// TIA Portal V20 export
VAR_GLOBAL   // PLC tag table "Spare"
   "BA010AZCRBK01.06" AT %I1000.6 : Bool;   // SPARE
   "BA010AZCRBK01.07" AT %I1000.7 : Bool;   // SPARE
   "BA010AZCRBK01.16" AT %I1001.6 : Bool;   // SPARE
   "BA010AZCRBK01.17" AT %I1001.7 : Bool;   // SPARE
   "BA010AZCRPM01.01" AT %Q2000.1 : Bool;   // SPARE
   "BA010AZCRPM01.03" AT %Q2000.3 : Bool;   // SPARE
   "BA010AZCRPM01.14" AT %Q2001.4 : Bool;   // SPARE
   "BA010AZCRPM01.15" AT %Q2001.5 : Bool;   // SPARE
   "BA010AZCRPM01.16" AT %Q2001.6 : Bool;   // SPARE
   "BA010AZCRPM01.17" AT %Q2001.7 : Bool;   // SPARE
   "BA010AZCRBK02.08" AT %I1005.0 : Bool;   // SPARE
   "BA010AZCRBK02.09" AT %I1005.1 : Bool;   // SPARE
   "BA010AZCRBK02.10" AT %I1005.2 : Bool;   // SPARE
   "BA010AZCRBK02.11" AT %I1005.3 : Bool;   // SPARE
   "BA010AZCRBK02.12" AT %I1005.4 : Bool;   // SPARE
   "BA010AZCRBK02.13" AT %I1005.5 : Bool;   // SPARE
   "BA010AZCRBK02.14" AT %I1005.6 : Bool;   // SPARE
   "BA010AZCRBK02.15" AT %I1005.7 : Bool;   // SPARE
   "BA010AZCRPM02.16" AT %Q2005.6 : Bool;   // SPARE
   "BA010AZCRPM02.17" AT %Q2005.7 : Bool;   // SPARE
   "BA010AZCRBK03.07" AT %I1008.7 : Bool;   // SPARE
   "BA010AZCRBK03.17" AT %I1009.7 : Bool;   // SPARE
   "BA010AZCRPM03.14" AT %Q2009.4 : Bool;   // SPARE
   "BA010AZCRPM03.15" AT %Q2009.5 : Bool;   // SPARE
   "BA010AZCRPM03.16" AT %Q2009.6 : Bool;   // SPARE
   "BA010AZCRPM03.17" AT %Q2009.7 : Bool;   // SPARE
   "BA010AZCRBK04.07" AT %I1012.7 : Bool;   // SPARE
   "BA010AZCRBK04.16" AT %I1013.6 : Bool;   // SPARE
   "BA010AZCRBK04.17" AT %I1013.7 : Bool;   // SPARE
   "BA010AZCRBK05.00" AT %I1016.0 : Bool;   // SPARE
   "BA010AZCRBK05.01" AT %I1016.1 : Bool;   // SPARE
   "BA010AZCRBK05.10" AT %I1017.0 : Bool;   // SPARE
   "BA010AZCRBK05.11" AT %I1017.1 : Bool;   // SPARE
   "BA010AZCRBK05.17" AT %I1017.7 : Bool;   // SPARE
   "BA010AZCRBK06.16" AT %I1021.6 : Bool;   // SPARE
   "BA010AZCRBK07.12" AT %I1025.2 : Bool;   // SPARE
   "BA010AZCRBK07.15" AT %I1025.5 : Bool;   // SPARE
   "BA010AZCRBK07.16" AT %I1025.6 : Bool;   // NG & MANUAL INPUT MAGAZINE FULL SENSOR EMITTER
   "BA010AZCRBK07.17" AT %I1025.7 : Bool;   // SPARE
   "BA010AZCRBK08.10" AT %Q2101.0 : Bool;   // SPARE
   "BA010AZCRBK08.11" AT %Q2101.1 : Bool;   // SPARE
   "BA010AZCRBK08.12" AT %Q2101.2 : Bool;   // SPARE
   "BA010AZCRBK08.13" AT %Q2101.3 : Bool;   // SPARE
   "BA010AZCRBK08.14" AT %Q2101.4 : Bool;   // SPARE
   "BA010AZCRBK08.15" AT %Q2101.5 : Bool;   // SPARE
   "BA010AZCRBK08.16" AT %Q2101.6 : Bool;   // SPARE
   "BA010AZCRBK08.17" AT %Q2101.7 : Bool;   // SPARE
   "BA010AZCRBK09.13" AT %Q2105.3 : Bool;   // SPARE
   "BA010AZCRBK09.14" AT %Q2105.4 : Bool;   // SPARE
   "BA010AZCRBK09.15" AT %Q2105.5 : Bool;   // SPARE
   "BA010AZCRBK09.16" AT %Q2105.6 : Bool;   // SPARE
   "BA010AZCRBK09.17" AT %Q2105.7 : Bool;   // SPARE
   "BA010AZCRSP504.01" AT %IW3110 : Int;   // SPARE
   "BA010AZCRSP504.02" AT %IW3112 : Int;   // SPARE
   "BA010AZCRSP504.03" AT %IW3114 : Int;   // SPARE
   "BA010AZCRSP505.01" AT %QW3202 : Int;   // SPARE
   "BA010AZCRSP505.02" AT %QW3204 : Int;   // SPARE
   "BA010AZCRSP505.03" AT %QW3206 : Int;   // SPARE
   "BA010AZCRSP507.03" AT %I3350.3 : Bool;   // SPARE
   "BA010AZCRSP501.02" AT %I3000.2 : Bool;   // SPARE
   "BA010AZCRSP501.03" AT %I3000.3 : Bool;   // SPARE
   "BA010AZCRSP501.06" AT %I3000.6 : Bool;   // SPARE
   "BA010AZCRSP501.07" AT %I3000.7 : Bool;   // SPARE
   "BA010AZCRSP501.10" AT %I3001.0 : Bool;   // SPARE
   "BA010AZCRSP501.11" AT %I3001.1 : Bool;   // SPARE
   "BA010AZCRSP501.12" AT %I3001.2 : Bool;   // SPARE
   "BA010AZCRSP501.13" AT %I3001.3 : Bool;   // SPARE
   "BA010AZCRSP501.14" AT %I3001.4 : Bool;   // SPARE
   "BA010AZCRSP501.15" AT %I3001.5 : Bool;   // SPARE
   "BA010AZCRSP501.16" AT %I3001.6 : Bool;   // SPARE
   "BA010AZCRSP501.17" AT %I3001.7 : Bool;   // SPARE
   "BA010AZCRSP502.00" AT %Q3000.0 : Bool;   // SPARE
   "BA010AZCRSP502.01" AT %Q3000.1 : Bool;   // SPARE
   "BA010AZCRSP502.02" AT %Q3000.2 : Bool;   // SPARE
   "BA010AZCRSP502.03" AT %Q3000.3 : Bool;   // SPARE
   "BA010AZCRSP502.04" AT %Q3000.4 : Bool;   // SPARE
   "BA010AZCRSP502.05" AT %Q3000.5 : Bool;   // SPARE
   "BA010AZCRSP502.06" AT %Q3000.6 : Bool;   // SPARE
   "BA010AZCRSP502.07" AT %Q3000.7 : Bool;   // SPARE
   "BA010AZCRSP502.10" AT %Q3001.0 : Bool;   // SPARE
   "BA010AZCRSP502.11" AT %Q3001.1 : Bool;   // SPARE
   "BA010AZCRSP502.12" AT %Q3001.2 : Bool;   // SPARE
   "BA010AZCRSP502.13" AT %Q3001.3 : Bool;   // SPARE
   "BA010AZCRSP502.14" AT %Q3001.4 : Bool;   // SPARE
   "BA010AZCRSP502.15" AT %Q3001.5 : Bool;   // SPARE
   "BA010AZCRSP502.16" AT %Q3001.6 : Bool;   // SPARE
   "BA010AZCRSP502.17" AT %Q3001.7 : Bool;   // SPARE
   "BA010AZCRBK07.14" AT %I1025.4 : Bool;   // ELECTRODE NG BOX FULL SENSOR EMITTER
   "BA010AZCRBK10.03" AT %Q2108.3 : Bool;   // SPARE
   "BA010AZCRBK10.04" AT %Q2108.4 : Bool;   // SPARE
   "BA010AZCRBK10.05" AT %Q2108.5 : Bool;   // SPARE
   "BA010AZCRBK10.06" AT %Q2108.6 : Bool;   // SPARE
   "BA010AZCRBK10.07" AT %Q2108.7 : Bool;   // SPARE
   "BA010AZCRBK09.10" AT %Q2105.0 : Bool;   // SPARE
   "BA010AZCRBK09.11" AT %Q2105.1 : Bool;   // SPARE
   "BA010AZCRBK09.12" AT %Q2105.2 : Bool;   // SPARE
   "BA010AZCRPM01.04" AT %Q2000.4 : Bool;   // SPARE
   "BA010AZCRPM01.05" AT %Q2000.5 : Bool;   // SPARE
   "BA010AZCRPM01.06" AT %Q2000.6 : Bool;   // SPARE
   "BA010AZCRPM01.07" AT %Q2000.7 : Bool;   // SPARE
   "BA010AZCRPM05.02" AT %Q2016.2 : Bool;   // SPARE
   "BA010AZCRPM05.03" AT %Q2016.3 : Bool;   // SPARE
   "BA010AZCRPM05.04" AT %Q2016.4 : Bool;   // SPARE
   "BA010AZCRPM05.05" AT %Q2016.5 : Bool;   // SPARE
   "BA010AZCRPM05.06" AT %Q2016.6 : Bool;   // SPARE
   "BA010AZCRPM05.07" AT %Q2016.7 : Bool;   // SPARE
   "BA010AZCRPM05.10" AT %Q2017.0 : Bool;   // SPARE
   "BA010AZCRPM05.11" AT %Q2017.1 : Bool;   // SPARE
   "BA010AZCRPM05.12" AT %Q2017.2 : Bool;   // SPARE
   "BA010AZCRPM05.13" AT %Q2017.3 : Bool;   // SPARE
   "BA010AZCRPM05.14" AT %Q2017.4 : Bool;   // SPARE
   "BA010AZCRPM05.15" AT %Q2017.5 : Bool;   // SPARE
   "BA010AZCRPM05.16" AT %Q2017.6 : Bool;   // SPARE
   "BA010AZCRPM05.17" AT %Q2017.7 : Bool;   // SPARE
   "BA010AZCRPM06.02" AT %Q2020.2 : Bool;   // SPARE
   "BA010AZCRPM06.03" AT %Q2020.3 : Bool;   // SPARE
   "BA010AZCRPM06.04" AT %Q2020.4 : Bool;   // SPARE
   "BA010AZCRPM06.05" AT %Q2020.5 : Bool;   // SPARE
   "BA010AZCRPM06.06" AT %Q2020.6 : Bool;   // SPARE
   "BA010AZCRPM06.07" AT %Q2020.7 : Bool;   // SPARE
   "BA010AZCRPM06.10" AT %Q2021.0 : Bool;   // SPARE
   "BA010AZCRPM06.11" AT %Q2021.1 : Bool;   // SPARE
   "BA010AZCRPM06.12" AT %Q2021.2 : Bool;   // SPARE
   "BA010AZCRPM06.13" AT %Q2021.3 : Bool;   // SPARE
   "BA010AZCRPM06.14" AT %Q2021.4 : Bool;   // SPARE
   "BA010AZCRPM06.15" AT %Q2021.5 : Bool;   // SPARE
   "BA010AZCRPM06.16" AT %Q2021.6 : Bool;   // SPARE
   "BA010AZCRPM06.17" AT %Q2021.7 : Bool;   // SPARE
END_VAR
